FUNCTION_BLOCK FB_Lag_filter
VAR_INPUT
	In: REAL;
	Time_const: TIME;
END_VAR
VAR_OUTPUT
	Out: REAL;
END_VAR
VAR	
	Scan_time: REAL;
	T: REAL;
END_VAR

Scan_time:= UINT_TO_REAL(_TaskInfo[1].CycleTime) / 10.0;
T:= TIME_TO_REAL(Time_const);

Out:= Out + (In - Out) * Scan_Time / (T - Scan_time);

END_FUNCTION_BLOCK

(* stored: Version 1.1.0.1, ProductVersion 3.1.4024.0
   POU FB_Lag_filter: Id {fc03950e-7a0e-4c4f-8e5e-e5c24060ece1}, SpecialFunc None *)
